// TwinCAT 3 PLC project ExtractorPLC
// ProgramVersion: 3.1.4024.0
// libraries:
//   Tc2_MC2, * (Beckhoff Automation GmbH)
//   Tc2_Standard, * (Beckhoff Automation GmbH)
//   Tc2_System, * (Beckhoff Automation GmbH)
//   Tc3_Module, * (Beckhoff Automation GmbH)
// project tree:
//   DUTs/ CL_Axis.TcPOU, E_AXIS_MOVE_PROFILE.TcDUT, E_StepAxis.TcDUT, ST_AXIS_MOVE_PROFILE.TcDUT
//   GVLs/ C.TcGVL, GAxes.TcGVL
//   / PlcTask.TcTTO
//   POUs/ CL_Debug.TcPOU, MAIN.TcPOU
// real-time tasks:
//   TASK PlcTask: cycle T#10ms, priority 20, ADS port 350
// motion (NC):
//   TASK NC-Task 1 SAF: cycle T#2ms, priority 4, ADS port 501
//   TASK NC-Task 1 SVB: cycle T#10ms, priority 8, ADS port 511
//   AXIS Axis 1 (id 1)
//     General: UnitName=m
//     Dynamic: AccelerationMaximum=98224.9365, DecelerationMaximum=98224.9365, Acceleration=982.25, Deceleration=982.25, Jerk=2946.75
//     Velo: RefSearch=40, RefSync=6.54833, SlowManual=32.74165, FastManual=196.4499, Fast=654.833, Maximum=654.833
//     OtherSettings: AllowMotionCmdToExtSetGenAxis=true
//     encoder EncType=19
//       EncPara: ScaleFactorNumerator=238.5, ScaleFactorDenominator=52428800, Inverse=true, MaxCount=#xffffffff
//         Inc: RefPosition=1.37, RefMode=1
//     drive DrvType=16
//       DrvPara: Inverse=true, MaxCount=#xffffffff, DriveControlDWord=#x00020100
//         Analog: VeloReferenz=720.3163, VeloScale=71.5255737304688, TorqueSetpointScale=10, ScaleFactorActTorque=0.1
//         TimeComp: TaskDelayCycles=1
//     controller CtrType=1
//       CtrPara: PriorControlFactor=1
//         Observer: BandWidth=20
// I/O:
//   DEVICE Device 1 (EtherCAT), AmsNetId 10.10.10.1.2.1
//     Term 1 (EK1200) [EK1200-5000 EtherCAT Power supply (2A E-Bus)]
//       Term 2 (EK1122) [EK1122 2 port EtherCAT junction]
//         AX8620 [AX8620-0000-0105]
//           AX8206 [AX8206-0200-0104 (2Ch. 6A servo axis, safe-motion)]
//             modules: Device, Device, Device, Device, Device, Device, Device, Device, Device, Device, Device (Safety), Device, Device, Device, Device, Device, Device, Device, Device, Device, Device, Device, Device, Device, Device, Device, Device, Device, Device, Device, Device, Ch A, Ch A, Ch A, Ch A, Ch A, Ch A, Ch A, Ch A, Ch A, Ch A, Ch A, Ch A, Ch A, Ch A, Ch A, Ch A, Ch A, Ch A, Ch A, Ch A, Ch A, Ch A, Ch A, Ch A, Ch A, Ch A, Ch A, Ch B, Ch B, Ch B, Ch B, Ch B, Ch B, Ch B, Ch B, Ch B, Ch B, Ch B, Ch B, Ch B, Ch B, Ch B, Ch B, Ch B, Ch B, Ch B, Ch B, Ch B, Ch B, Ch B, Ch B, Ch B, Ch B
//             startup 12992:1 := 414D383032312D78427830 // Ch A Motor parameters / Configured motor type
//             startup 24768:0 := FEFF // Ch A Interpolation sub mode select
//             startup 13000:5 := 0200 // Ch A Motor thermal model / Reaction
//             startup 13000:6 := 0000C841 // Ch A Motor thermal model / Partial fraction factor
//             startup 12992:12 := 0000FA45 // Ch A Motor parameters / Motor rated speed
//             startup 12992:13 := C9E5FF3E // Ch A Motor parameters / Motor rated torque
//             startup 24694:0 := F4010000 // Ch A Motor standstill torque
//             startup 24800:0 := D007 // Ch A Positive torque/force limit value
//             startup 24801:0 := D007 // Ch A Negative torque/force limit value
//             startup 12288:6 := 4158383230362D303230302D30303030 // Ch A AxisMain parameters / Configured drive type
//             startup 12867:1 := 9A99593F // Ch A TorqueCtrl parameters / Configured channel rated current
//             startup 12867:2 := 33332340 // Ch A TorqueCtrl parameters / Configured channel peak current
//             startup 24672:0 := 08 // Ch A Modes of operation
//             startup 12864:1 := 0D4D7043 // Ch A TorqueCtrl parameters mappable / Torque control proportional gain q
//             startup 12864:2 := 8A0E7C39 // Ch A TorqueCtrl parameters mappable / Torque control integral action time q
//             startup 12608:1 := FBD1CD3B // Ch A VeloCtrl parameters mappable / Velocity control proportional gain
//             startup 12608:2 := 6F12033C // Ch A VeloCtrl parameters mappable / Velocity control integral action time
//             startup 12608:3 := 00203246 // Ch A VeloCtrl parameters mappable / Bipolar velocity limit value
//             startup 12992:15 := 0100 // Ch A Motor parameters / Motor temperature sensor connection
//             startup 12611:4 := 0400 // Ch A VeloCtrl observer / Observer type
//             startup 24672:0 := 08 // Ch A Modes of operation
//             startup 12296:2 := 00 // Ch A AxisMain parameters encoder polarity / Primary encoder actual values
//           Term 5 (EL9011) [EL9011 End Terminal]
// variable links:
//   (this object) <-> Device 1 (EtherCAT)/Term 1 (EK1200)/Term 2 (EK1122)/AX8620/AX8206
//     Drive/Inputs/In/nDataIn1 <-> Ch A/Ch A PositionControl Inputs/Ch A Following error actual value
//     Drive/Inputs/In/nDataIn3[0] <-> Ch A/Ch A TorqueControl Inputs/Ch A Torque/force actual value
//     Drive/Inputs/In/nDcOutputTime <-> InfoData/DcOutputShift
//     Drive/Inputs/In/nState1 <-> Ch A/Ch A AxisMain Inputs/Ch A Statusword
//     Drive/Inputs/In/nState2 <-> Ch A/Ch A AxisMain Inputs/Ch A Statusword @bit 8
//     Drive/Inputs/In/nState4 @bit 1 <-> Ch B/WcState/InputToggle0
//     Drive/Inputs/In/nState4 <-> Ch B/WcState/WcState0
//     Drive/Outputs/Out/nCtrl1 <-> Ch A/Ch A AxisMain Outputs/Ch A Controlword
//     Drive/Outputs/Out/nCtrl2 <-> Ch A/Ch A AxisMain Outputs/Ch A Controlword @bit 8
//     Drive/Outputs/Out/nDataOut1 <-> Ch A/Ch A Interpolator Outputs/Ch A Target position
//     Drive/Outputs/Out/nDataOut2 <-> Ch A/Ch A Interpolator Outputs/Ch A Target velocity
//     Enc/Inputs/In/nDataIn1 <-> Ch A/Ch A AxisMain Inputs/Ch A Position actual value
//     Enc/Inputs/In/nDcInputTime <-> InfoData/DcInputShift
//     Enc/Inputs/In/nState2 @bit 5 <-> Ch A/Ch A AxisMain Inputs/Position actual value invalid
//     Enc/Inputs/In/nState4 @bit 1 <-> Ch B/WcState/InputToggle0
//     Enc/Inputs/In/nState4 <-> Ch B/WcState/WcState0
//   (this object) <-> Device 1 (EtherCAT)
//     Term 1 (EK1200)/Term 2 (EK1122)/AX8620/AX8206/Device/DeviceMain Outputs/Power supply controlword <-> Term 1 (EK1200)/Term 2 (EK1122)/AX8620/PSM Controlword for axis/Controlword for axis
//     Term 1 (EK1200)/Term 2 (EK1122)/AX8620/PSM Controlword for axis/Controlword for axis <-> Term 1 (EK1200)/Term 2 (EK1122)/AX8620/AX8206/Device/DeviceMain Outputs/Power supply controlword
//   ExtractorPLC Instance <-> Device 1 (EtherCAT)/Term 1 (EK1200)/Term 2 (EK1122)/AX8620/AX8206
//     PlcTask Inputs/GAxes.nTorqueForce <-> Ch A/Ch A TorqueControl Inputs/Ch A Torque/force actual value
//     PlcTask Inputs/GAxes.udHomingSensor <-> Ch A/Ch A AxisMain Inputs/Ch A Digital inputs
//   ExtractorPLC Instance <-> NC-Task 1 SAF/Axes/Axis 1
//     PlcTask Inputs/GAxes.ExtractorAxis.NcToPlc <-> Outputs/ToPlc
//     PlcTask Outputs/GAxes.ExtractorAxis.PlcToNc <-> Inputs/FromPlc

CONFIGURATION ExtractorPLC
    RESOURCE PLC ON TwinCAT3
        TASK PlcTask(INTERVAL := T#10ms, PRIORITY := 20);
        PROGRAM MAIN WITH PlcTask : MAIN;
    END_RESOURCE
END_CONFIGURATION

// ---- DUTs/E_AXIS_MOVE_PROFILE.TcDUT
(*
Description:
Enum of moving profiles possibilities
Created by 	: BRU
Creation    : xx.11.2021	
$Author: dbruegger $
$Date: 2021-11-18 16:38:14 +0100 (jeu., 18 nov. 2021) $
$Revision: 155 $
*)
{attribute 'qualified_only'}
{attribute 'strict'}
TYPE E_AXIS_MOVE_PROFILE :
(
	Slow	:= 0,
	Nominal	:= 1,
	Fast	:= 2// Don't increase this without increase size of all arrays used this enum!!!!!!!!!!!
)INT;
END_TYPE

// ---- DUTs/E_StepAxis.TcDUT
{attribute 'qualified_only'}
{attribute 'strict'}
TYPE E_StepAxis :
(
	Idle	        := 0,
	// STEPS POWER
	PoweringOn		:= 2,
	PoweringOff	  := 4,
	
	// STEPS ABSOLUTE
  InitMoveAbs   := 10,
	MoveAbs		    := 11,
	EndMoveAbs    := 12,
  
	// STEPS STOP
  InitStop      := 50,
	Stopping		  := 51,
  EndStopping   := 52,
	
	// STEPS HOMING
  InitHoming    := 60,
	Homing			  := 61,
  EndHoming     := 62,
  InitAbortHoming := 63,
  AbortHoming   := 64,
  InitRetryHoming := 65,
  RetryHoming     := 66,
  
	
	// STEPS Reset
  InitReset     := 70,
	Resetting		  := 71,
  EndReset      := 72,
	
	// STEPS ERROR
	ERROR			    := 100
);
END_TYPE

// ---- DUTs/ST_AXIS_MOVE_PROFILE.TcDUT
(*
Description:
Structur of a moving profile
Created by 	: BRU
Creation    : xx.11.2021	
$Author: dbruegger $
$Date: 2021-11-18 16:38:14 +0100 (jeu., 18 nov. 2021) $
$Revision: 155 $
*)
TYPE ST_AXIS_MOVE_PROFILE :
STRUCT
	Velo	: REAL;// Velocity
	Acc		: REAL;// Acceleration
	Dec		: REAL;// Deceleration
	Jerk	: REAL;// Jerk
END_STRUCT
END_TYPE

// ---- GVLs/C.TcGVL
{attribute 'qualified_only'}
VAR_GLOBAL CONSTANT 
	//debug
	uiHistoStep_C								        : INT := 50;
END_VAR

// ---- GVLs/GAxes.TcGVL
VAR_GLOBAL
  {attribute 'TcNcAxis' := 'Axis 1'} 
  ExtractorAxis		      :  AXIS_REF;
  
  {attribute 'TcLinkTo' := 'TIIB[AX8620]^AX8206^Ch A^Ch A AxisMain Inputs^Ch A Digital inputs;'}
  udHomingSensor AT %I* : UDINT;
  
  {attribute 'TcLinkTo' := 'TIIB[AX8620]^AX8206^Ch A^Ch A TorqueControl Inputs^Ch A Torque/force actual value;'}
  nTorqueForce AT %I*   : INT;
END_VAR

// ---- POUs/MAIN.TcPOU
PROGRAM MAIN
VAR
  cnt             : DINT;
  nStep           : INT :=0;
  objAxis         : CL_Axis;
  nLineNumber     : INT;
  lrOffsetHoming  : LREAL := -180;
END_VAR

objAxis();
CASE nStep OF
  0 : 
    objAxis.SetAxisProfile(Profile := E_AXIS_MOVE_PROFILE.Slow, Velocity := 100, Acceleration := 1000, Deceleration := 1000, Jerk := 10000);
    objAxis.SetAxisProfile(Profile := E_AXIS_MOVE_PROFILE.Nominal, Velocity := 200, Acceleration := 1000, Deceleration := 1000, Jerk := 10000);
    objAxis.SetAxisProfile(Profile := E_AXIS_MOVE_PROFILE.Fast, Velocity := 900, Acceleration := 2000, Deceleration := 2000, Jerk := 20000);
    objAxis.Init(bHomingSensor_P := ADR(GAxes.udHomingSensor.19),nLineNumber_P := ADR(nLineNumber),nAxisTorque_P := ADR(GAxes.nTorqueForce),AxisREF_P := ADR(GAxes.ExtractorAxis));
    nStep := 10;
  10: 
    objAxis.RequestPowerON();
    IF objAxis.bIsBusy THEN
      nStep := 20;
		END_IF
  20:
    IF NOT objAxis.bIsBusy AND objAxis.bIsPowered THEN
      nStep := 30;
		END_IF
  30:
    objAxis.RequestHoming(lrOffsetHoming);
    IF objAxis.bIsBusy THEN
      nStep := 40;
		END_IF
  40:
    IF NOT objAxis.bIsBusy AND objAxis.bIsHomed THEN
      nStep := 50;
		END_IF    
    
  50:
    objAxis.RequestMove(Profile:= E_AXIS_MOVE_PROFILE.Fast,Target := 400); 
    IF objAxis.bIsBusy THEN
      nStep := 60;    
		END_IF   
  60: 
    IF NOT objAxis.bIsBusy THEN
      nStep := 70;       
		END_IF  
  70:
    objAxis.RequestMove(Profile:= E_AXIS_MOVE_PROFILE.Fast,Target := -350); 
    IF objAxis.bIsBusy THEN
      nStep := 80;    
		END_IF   
  80: 
    IF NOT objAxis.bIsBusy THEN
      cnt := cnt + 1; 
      nStep := 50;       
		END_IF  
    
 999: nStep := 999;
END_CASE

END_PROGRAM

// ---- DUTs/CL_Axis.TcPOU
FUNCTION_BLOCK CL_Axis EXTENDS CL_Debug
VAR_INPUT
	bEnableMove     : BOOL := TRUE;   // Enable the moving of axis
	lrAxisOverride	: LREAL:= 100;    // Override of the axis
END_VAR
VAR_OUTPUT	
	bError			: BOOL := FALSE;
	nErrorId		: UDINT;
END_VAR
VAR
//  INTERNAL VAR
  _AxisREF_P		        		: POINTER TO AXIS_REF;
  _udCalibrationSensor_P  	: POINTER TO UDINT;
  _LineNumber_P             : POINTER TO INT;
  _nAxisTorque_P            : POINTER TO INT;
	_bIsDone                	: BOOL;
  _bIsBusy                	: BOOL;
  _lrActPos                 : LREAL;

//  Request var	BOOL
	bRequestStop		  				: BOOL := FALSE;
	bRequestPowerOn						: BOOL := FALSE;
	bRequestPowerOff					: BOOL := FALSE;
	bRequestHoming						: BOOL := FALSE;
	bRequestReset		  				: BOOL := FALSE;
	bRequestMoveAbso					: BOOL := FALSE;
	bInit               			: BOOL := FALSE;
	
// FBs
	fbPower				      : MC_Power;
	fbStop				      : MC_Stop;
	fbReset				      : MC_Reset; 
	fbHome				      : MC_Home;
  fbHomeInv				    : MC_Home;
	fbMoveAbso				  : MC_MoveAbsolute;
  fbReadStatus        : MC_ReadStatus;
  fbMoveJog           : MC_Jog;
  fbTimeRetryHomming  : TON := (PT := T#1S);
  fbTimeAbortHoming   : ton := (PT := T#20S);
  fbTrigErrorMotor    : R_Trig;
  
//Other var
	nStep			          : INT;
  
  stHomingOption	    : ST_HomingOptions;
  stHomingInvOption	  : ST_HomingOptions;
  //stJogControl        : ST_HmiControlMotor;
  lrSetHomingCheckPos : LREAL;
	lrnOffsetExtractorHoming : LREAL;

//Request var
	eRequestedProfile		: E_AXIS_MOVE_PROFILE := E_AXIS_MOVE_PROFILE.Slow;
	rRequestedTarget		: LREAL := 0;
	Profile				    	: ARRAY[0..2]OF ST_AXIS_MOVE_PROFILE ;
END_VAR

IF NOT bInit THEN
  RETURN;
END_IF

//CALL BLOCK
fbPower(Axis:= _AxisREF_P^, Override:= lrAxisOverride);
fbStop(Axis:= _AxisREF_P^);
fbReset(Axis:= _AxisREF_P^);
fbHome( Axis:= _AxisREF_P^, bCalibrationCam:=_udCalibrationSensor_P^.19,
		    Options := stHomingOption, Position := lrnOffsetExtractorHoming);
fbHomeInv( Axis:= _AxisREF_P^, bCalibrationCam:=_udCalibrationSensor_P^.19,
		    Options := stHomingInvOption, Position := lrnOffsetExtractorHoming);
fbMoveAbso(Axis:= _AxisREF_P^);
fbReadStatus(Axis:= _AxisREF_P^,Enable := TRUE);
//fbMoveJog(Axis := _AxisREF_P^,JogForward := stJogControl.bMoveFW, JogBackwards := stJogControl.bMoveBW);
fbTimeRetryHomming(IN := nStep = E_StepAxis.AbortHoming);
fbTimeAbortHoming(IN := nStep = E_StepAxis.RetryHoming);
fbTrigErrorMotor(CLK := _AxisREF_P^.NcToPlc.ErrorCode <> 0);
_lrActPos := _AxisREF_P^.NcToPlc.ActPos;


IF fbTrigErrorMotor.Q THEN
  nStep := E_StepAxis.Idle;
  bRequestMoveAbso := FALSE;
  bRequestHoming := FALSE;
  fbHome.Execute := FALSE;
  fbHomeInv.Execute := FALSE;
  fbMoveAbso.Execute := FALSE;
END_IF

// If bEnableMove is down, do a stop automatically
//IF NOT bEnableMove THEN
//	bRequestStop		:= TRUE;
//	eRequestedProfile	:= E_AXIS_MOVE_PROFILE.Fast;
//END_IF


CASE nStep OF
	// ------------------------------------------------------------------
	E_StepAxis.IDLE :	
		bRequestStop	:= FALSE;			
    IF bRequestPowerOff THEN
      nStep := E_StepAxis.PoweringOff;
      bRequestPowerOff	:= FALSE;
    ELSIF bRequestPowerOn THEN
      nStep := E_StepAxis.PoweringOn;
      bRequestPowerOn		:= FALSE;
    ELSIF bRequestMoveAbso THEN
      nStep := E_StepAxis.InitMoveAbs;
      bRequestMoveAbso	:= FALSE;
    ELSIF bRequestHoming THEN
      bRequestHoming		:= FALSE;
			IF _udCalibrationSensor_P^.19 THEN
				nStep := E_StepAxis.InitRetryHoming;
			ELSE
				nStep := E_StepAxis.InitHoming;
			END_IF	
    ELSIF bRequestReset OR (_AxisREF_P^.NcToPlc.ErrorCode <> 0) THEN
			//added to support MDF extractor: homing in both direction		
			nStep := E_StepAxis.InitReset;
      bRequestReset		:= FALSE;
    END_IF
	
	// ******************************************************************
	// --- POWER ---
	// ******************************************************************
		// ------------------------------------------------------------------
		E_StepAxis.PoweringOff :
      fbPower.Enable := FALSE;
			//objHommingError.Set(Activate:= FALSE);
      IF NOT fbPower.Status THEN
        _bIsDone	:= TRUE;
        _bIsBusy	:= FALSE;
        nStep := E_StepAxis.IDLE;
      ELSIF fbPower.Error THEN
        nErrorId := fbPower.ErrorID;
        nStep := E_StepAxis.ERROR;
      END_IF
			
		// ------------------------------------------------------------------
		E_StepAxis.PoweringOn :
      fbPower.Enable			:= TRUE;
      fbPower.Enable_Positive	:= TRUE;
      fbPower.Enable_Negative	:= TRUE;
      IF fbPower.Status THEN
        _bIsDone	:= TRUE;
        _bIsBusy	:= FALSE;
        nStep  := E_StepAxis.Idle;
      ELSIF fbPower.Error THEN
        fbPower.Enable			:= FALSE;
        fbPower.Enable_Positive	:= FALSE;
        fbPower.Enable_Negative	:= FALSE;
        _bIsBusy	:= FALSE;
        nStep  := E_StepAxis.Idle;      
      END_IF
			
	// ******************************************************************
	// --- ABSOLUTE ---
	// ******************************************************************
		// ------------------------------------------------------------------
		E_StepAxis.InitMoveAbs:
      fbMoveAbso.Position		:= rRequestedTarget;
      fbMoveAbso.Velocity		:= Profile[eRequestedProfile].Velo;
      fbMoveAbso.Acceleration	:= Profile[eRequestedProfile].Acc;
      fbMoveAbso.Deceleration	:= Profile[eRequestedProfile].Dec;
      fbMoveAbso.Jerk			:= Profile[eRequestedProfile].Jerk;
      fbMoveAbso.Execute			:= TRUE;
      IF fbMoveAbso.Busy THEN
         nStep := E_StepAxis.MoveAbs;
      END_IF
    
    // ------------------------------------------------------------------  
    E_StepAxis.MoveAbs:    
      IF fbMoveAbso.Done THEN
        nStep:= E_StepAxis.EndMoveAbs;
      ELSIF bRequestStop THEN
        fbMoveAbso.Execute := FALSE;
        nStep:= E_StepAxis.InitStop;
        bRequestStop := FALSE;
      ELSIF fbMoveAbso.Error THEN
        fbMoveAbso.Execute	:= false;
        _bIsBusy	:= FALSE;
        nStep     := E_StepAxis.Idle;
      END_IF
     
    // ------------------------------------------------------------------  
    E_StepAxis.EndMoveAbs: 
      _bIsDone	:= TRUE;
      _bIsBusy	:= FALSE;
      fbMoveAbso.Execute  := FALSE;
      nStep     := E_StepAxis.Idle;
						
	// ******************************************************************
	// --- STOP ---
	// ******************************************************************
		// ------------------------------------------------------------------
		E_StepAxis.InitStop :
			bRequestStop	:= FALSE;
      fbStop.Deceleration	:= Profile[eRequestedProfile].Dec;
      fbStop.Jerk			    := Profile[eRequestedProfile].Jerk;
      fbStop.Execute		  := TRUE;
      IF fbStop.Busy THEN
        nStep := E_StepAxis.Stopping;
			END_IF
                  
		// ------------------------------------------------------------------
		E_StepAxis.Stopping :        
      IF _AxisREF_P^.Status.NotMoving THEN
        _bIsDone	:= TRUE;
        _bIsBusy	:= FALSE;
        nStep  := E_StepAxis.EndStopping;
      END_IF
        
		// ------------------------------------------------------------------
		E_StepAxis.EndStopping :        
      fbStop.Execute	:= FALSE;
      //objHommingError.Set(Activate:= FALSE);
			nStep           := E_StepAxis.Idle;

	// ******************************************************************
	// --- HOMING ---
	// ******************************************************************
		// ------------------------------------------------------------------
		E_StepAxis.InitHoming:
      fbHome.Execute			:= TRUE;
      IF fbHome.Busy THEN
        nStep := E_StepAxis.Homing;
			END_IF      
    
    // ------------------------------------------------------------------  
    E_StepAxis.Homing:    
      IF fbHome.Done THEN
        nStep:= E_StepAxis.EndHoming;
      ELSIF bRequestStop THEN
        fbHome.Execute			:= false;
        nStep:= E_StepAxis.InitStop;
        bRequestStop := FALSE;
      ELSIF _nAxisTorque_P^ < -800  THEN
        nStep:= E_StepAxis.InitAbortHoming;    
      END_IF
 
		// ------------------------------------------------------------------
		E_StepAxis.InitAbortHoming:
      fbStop.Deceleration	:= Profile[eRequestedProfile].Dec;
      fbStop.Jerk			    := Profile[eRequestedProfile].Jerk;
      fbStop.Execute		  := TRUE;
      fbHome.Execute			:= FALSE;
      IF fbStop.Busy THEN
        nStep := E_StepAxis.AbortHoming;
			END_IF
      
		// ------------------------------------------------------------------
		E_StepAxis.AbortHoming:
      IF _AxisREF_P^.Status.NotMoving AND fbTimeRetryHomming.Q THEN
        fbStop.Execute	:= FALSE;
        nStep  := E_StepAxis.InitRetryHoming;
      END_IF    
    
    // ------------------------------------------------------------------  
    E_StepAxis.EndHoming: 
      _bIsDone	:= TRUE;
      _bIsBusy	:= FALSE;
      fbHome.Execute			:= FALSE;
      fbHomeInv.Execute			:= FALSE;
      nStep                   := E_StepAxis.Idle;
    
    // ------------------------------------------------------------------   
		E_StepAxis.InitRetryHoming:
      fbHomeInv.Execute			:= TRUE;
      IF fbHomeInv.Busy THEN
        lrSetHomingCheckPos := _AxisREF_P^.NcToPlc.ActPos;
        nStep := E_StepAxis.RetryHoming;
			END_IF  

    // ------------------------------------------------------------------  
    E_StepAxis.RetryHoming:    
      IF fbHomeInv.Done THEN
        nStep:= E_StepAxis.EndHoming;
      ELSIF bRequestStop THEN
        fbHomeInv.Execute			:= FALSE;
        nStep:= E_StepAxis.InitStop;
        bRequestStop := FALSE;
      ELSIF  (_nAxisTorque_P^ > 600) THEN
        nStep:= E_StepAxis.InitStop;
        fbHomeInv.Execute := FALSE;
        //objHommingError.Set(Activate:= TRUE);      
      END_IF
			
	// ******************************************************************
	// --- RESETTING ---
	// ******************************************************************
  	// ------------------------------------------------------------------
		E_StepAxis.InitReset :
      fbReset.Execute		:= TRUE;
      IF fbReset.Busy THEN
        nStep := E_StepAxis.Resetting;
      END_IF
      
    // ------------------------------------------------------------------
		E_StepAxis.Resetting :
      IF fbReset.Done THEN
        bError	:= FALSE;
        _bIsDone	:= TRUE;
        _bIsBusy	:= FALSE;
        nStep := E_StepAxis.EndReset;
      END_IF
      
		// ------------------------------------------------------------------
		E_StepAxis.EndReset:
      fbReset.Execute	:= FALSE;
      nStep := E_StepAxis.Idle;
			
	// ******************************************************************
	// --- ERROR ---
	// ******************************************************************
		// ------------------------------------------------------------------
		E_StepAxis.ERROR :
				//added by Tristan 23-4-2024
				fbPower.Enable			:= FALSE;
        fbPower.Enable_Positive	:= FALSE;
        fbPower.Enable_Negative	:= FALSE;
				      fbHome.Execute			:= FALSE;
      fbHomeInv.Execute			:= FALSE;
			bRequestStop := FALSE;
      bError	:= TRUE;
      _bIsBusy	:= FALSE;
END_CASE

// Call again to refresh cmd
fbPower(Axis:= _AxisREF_P^, Override:= lrAxisOverride);
fbStop(Axis:= _AxisREF_P^);
fbReset(Axis:= _AxisREF_P^);
fbHome( Axis:= _AxisREF_P^, bCalibrationCam:=_udCalibrationSensor_P^.19,
		    Options := stHomingOption, Position := lrnOffsetExtractorHoming);
fbHomeInv( Axis:= _AxisREF_P^, bCalibrationCam:=_udCalibrationSensor_P^.19,
		    Options := stHomingInvOption, Position := lrnOffsetExtractorHoming);
fbMoveAbso(Axis:= _AxisREF_P^);
fbReadStatus(Axis:= _AxisREF_P^,Enable := TRUE);

Case01Histo( nStep);

PROPERTY bIsBusy : bool
GET
bIsBusy := _bIsBusy;
END_GET
END_PROPERTY

PROPERTY bIsDone : bool
GET
bIsDone := _bIsDone;
END_GET
END_PROPERTY

PROPERTY bIsHomed : bool
GET
IF _AxisREF_P <> 0 THEN
	bIsHomed := _AxisREF_P^.Status.Homed;
END_IF
END_GET
END_PROPERTY

PROPERTY bIsInPos : bool
GET
bIsInPos := _AxisREF_P^.Status.InPositionArea;
END_GET
END_PROPERTY

PROPERTY bIsPowered : bool
GET
bIsPowered :=  fbPower.Status;
END_GET
END_PROPERTY

PROPERTY bIsStopped : BOOL
GET
bIsStopped := _AxisREF_P^.Status.NotMoving;
END_GET
END_PROPERTY

PROPERTY InError : bool
GET
InError := _AxisREF_P^.NcToPlc.ErrorCode <> 0;
END_GET
END_PROPERTY

METHOD Init : BOOL
VAR_INPUT
	AxisREF_P				      	: POINTER TO AXIS_REF;
  bHomingSensor_P			    : POINTER TO BOOL;
  nAxisTorque_P           : POINTER TO INT;
  nLineNumber_P           : POINTER TO INT;
END_VAR
IF NOT bInit and nAxisTorque_P <> 0 AND bHomingSensor_P <> 0 AND nLineNumber_P <> 0 AND AxisREF_P <> 0 THEN
  bInit := TRUE;

	_udCalibrationSensor_P := bHomingSensor_P;
	_AxisREF_P := AxisREF_P;
	_LineNumber_P := nLineNumber_P;
	_nAxisTorque_P :=  nAxisTorque_P;
	
	stHomingOption.SearchDirection := MC_Direction.MC_Negative_Direction;
	stHomingOption.SyncDirection := MC_Direction.MC_Positive_Direction;
	stHomingInvOption.SearchDirection := MC_Direction.MC_Positive_Direction;
	stHomingInvOption.SyncDirection := MC_Direction.MC_Positive_Direction;
END_IF
END_METHOD

PROPERTY lrActPos : lreal
GET
lrActPos := _lrActPos;
END_GET
END_PROPERTY

PROPERTY lrActTorque : lreal
GET
lrActTorque := _AxisREF_P^.NcToPlc.ActTorque;
END_GET
END_PROPERTY

{attribute 'TcRpcEnable'}
METHOD RequestHoming : bool
VAR_INPUT
	lrnOffsetExtractorHomingRef : LREAL;
END_VAR
_bIsDone			:= FALSE;
IF bIsPowered AND bEnableMove AND NOT bError THEN
	bRequestHoming 		:= TRUE;
	_bIsBusy				    := TRUE;
	lrnOffsetExtractorHoming := lrnOffsetExtractorHomingRef;
END_IF
END_METHOD

{attribute 'TcRpcEnable'}
METHOD RequestMove : BOOL
VAR_INPUT
	Profile	: E_AXIS_MOVE_PROFILE;
	Target	: LREAL;
END_VAR
_bIsDone		:= FALSE;

IF bIsPowered AND bEnableMove AND NOT bError AND NOT bIsBusy THEN
  _bIsBusy				  := TRUE;
  bRequestMoveAbso	:= TRUE;
  eRequestedProfile	:= Profile;
  rRequestedTarget	:= Target;
END_IF
END_METHOD

{attribute 'TcRpcEnable'}
METHOD RequestPowerOFF : BOOL
VAR_INPUT
END_VAR
_bIsDone			:= FALSE;

IF bIsPowered AND NOT bIsBusy THEN
	bRequestPowerOFF	:= TRUE;
	_bIsBusy				:= TRUE;
END_IF
END_METHOD

{attribute 'TcRpcEnable'}
METHOD RequestPowerON : bool
VAR_INPUT
END_VAR
_bIsDone			:= FALSE;

IF NOT bIsPowered AND NOT bError THEN
	bRequestPowerON		:= TRUE;
	_bIsBusy				  := TRUE;
END_IF
END_METHOD

{attribute 'TcRpcEnable'}
METHOD RequestReset :bool
VAR_INPUT
END_VAR
_bIsDone			:= FALSE;

IF TRUE(*bError*) THEN
	bRequestReset 		:= TRUE;
	_bIsBusy				:= TRUE;
	nErrorId			:= 0;
END_IF
END_METHOD

{attribute 'TcRpcEnable'}
METHOD RequestStop : bool
VAR_INPUT
	Profile	: E_AXIS_MOVE_PROFILE;
END_VAR
_bIsDone		:= FALSE;
IF _bIsBusy THEN
	bRequestStop := TRUE;
	eRequestedProfile	:= Profile;
END_IF
END_METHOD

{attribute 'TcRpcEnable'}
METHOD SetAxisProfile : BOOL
VAR_INPUT
	Profile			: E_AXIS_MOVE_PROFILE;
	Velocity		: REAL;
	Acceleration	: REAL;
	Deceleration	: REAL;
	Jerk			: REAL;
END_VAR
THIS^.Profile[Profile].Velo		:= Velocity;
THIS^.Profile[Profile].Acc		:= Acceleration;
THIS^.Profile[Profile].Dec		:= Deceleration;
THIS^.Profile[Profile].Jerk		:= Jerk;
END_METHOD

END_FUNCTION_BLOCK

// ---- POUs/CL_Debug.TcPOU
FUNCTION_BLOCK CL_Debug
VAR
	i01                         : INT;
  nHistoryStep_AR01           : ARRAY[0..C.uiHistoStep_C] OF DINT;
  nLastStep01                 : DINT := -1;
  
  i02                         : INT;
  nHistoryStep_AR02           : ARRAY[0..C.uiHistoStep_C] OF DINT;
  nLastStep02                 : DINT := -1;
  
  i03                         : INT;
  nHistoryStep_AR03           : ARRAY[0..C.uiHistoStep_C] OF DINT;
  nLastStep03                 : DINT := -1;
END_VAR

METHOD Case01Histo : BOOL
VAR_INPUT
	nStep : DINT;
END_VAR
IF nStep <> nLastStep01 THEN
  nLastStep01 := nStep;
  FOR i01:= C.uiHistoStep_C TO 1 BY -1 DO
    nHistoryStep_AR01[i01] := nHistoryStep_AR01[i01-1];
  END_FOR
  nHistoryStep_AR01[0] := nStep;
END_IF
END_METHOD

METHOD Case02Histo : BOOL
VAR_INPUT
	nStep : DINT;
END_VAR
IF nStep <> nLastStep02 THEN
  nLastStep02 := nStep;
  FOR i02:= C.uiHistoStep_C TO 1 BY -1 DO
    nHistoryStep_AR02[i02] := nHistoryStep_AR01[i02-1];
  END_FOR
  nHistoryStep_AR02[0] := nStep;
END_IF
END_METHOD

METHOD Case03Histo : BOOL
VAR_INPUT
	nStep : DINT;
END_VAR
IF nStep <> nLastStep03 THEN
  nLastStep03 := nStep;
  FOR i03:= C.uiHistoStep_C TO 1 BY -1 DO
    nHistoryStep_AR03[i03] := nHistoryStep_AR01[i03-1];
  END_FOR
  nHistoryStep_AR03[0] := nStep;
END_IF
END_METHOD

END_FUNCTION_BLOCK
